FUNCTION_BLOCK BasicCalcEmptyAlgs (* Basic FB with empty ECC *)
  (* Standard: 61499-2 *)
  (* Version 1.0, 2023-07-26, AK115394 *)
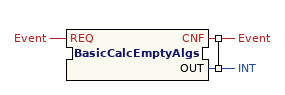
  EVENT_INPUT
    REQ;
  END_EVENT
  EVENT_OUTPUT
    CNF WITH OUT;
  END_EVENT
  VAR_OUTPUT
    OUT : INT;
  END_VAR
  VAR
    Fn0 : INT;
    Fn1 : INT;
    Fnx : INT;
  END_VAR
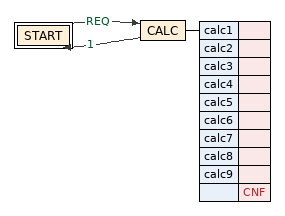
  EC_STATES
    START; (* Initial State *)
    CALC : calc1, calc2, calc3, calc4, calc5, calc6, calc7, calc8, calc9, -> CNF;
  END_STATES
  EC_TRANSITIONS
    START TO CALC := REQ;
    CALC TO START := 1;
  END_TRANSITIONS
  ALGORITHM calc1 IN ST:
 OUT:=1+1;
  END_ALGORITHM
  ALGORITHM calc2 IN ST:
 OUT:=2+2;
  END_ALGORITHM
  ALGORITHM calc3 IN ST:
 OUT:=3+3;
  END_ALGORITHM
  ALGORITHM calc4 IN ST:
 OUT:=4+4;
  END_ALGORITHM
  ALGORITHM calc5 IN ST:
 OUT:=5+5;
  END_ALGORITHM
  ALGORITHM calc6 IN ST:
 OUT:=6+6;
  END_ALGORITHM
  ALGORITHM calc7 IN ST:
 OUT:=7+7;
  END_ALGORITHM
  ALGORITHM calc8 IN ST:
 OUT:=8+8;
  END_ALGORITHM
  ALGORITHM calc9 IN ST:
 OUT:=9+9;
  END_ALGORITHM
END_FUNCTION_BLOCK
